PROGRAM Axis06_Status
VAR
//System_Bit
	Always_ON	:	BOOL	:=TRUE	;//상시 ON 
	Always_OFF	:	BOOL	:=FALSE	;//상시 OFF
	
	Real_Position_Data : ARRAY[0..39999] OF LREAL; // 40,000개 데이터 저장 (2초 보장)
    nIndex          : DINT := 0;                // 배열 인덱스 (0 ~ 39999)

	Axis06_Position_Read: MC_ReadActualPosition;
	Axis06_Velocity_Read: MC_ReadActualVelocity;
	nCounter: INT;
	i: INT;
	Test04: BOOL;
	Test05: BOOL;
	TEST005: BOOL;
	Axis06_Reset_01: MC_Reset;
END_VAR

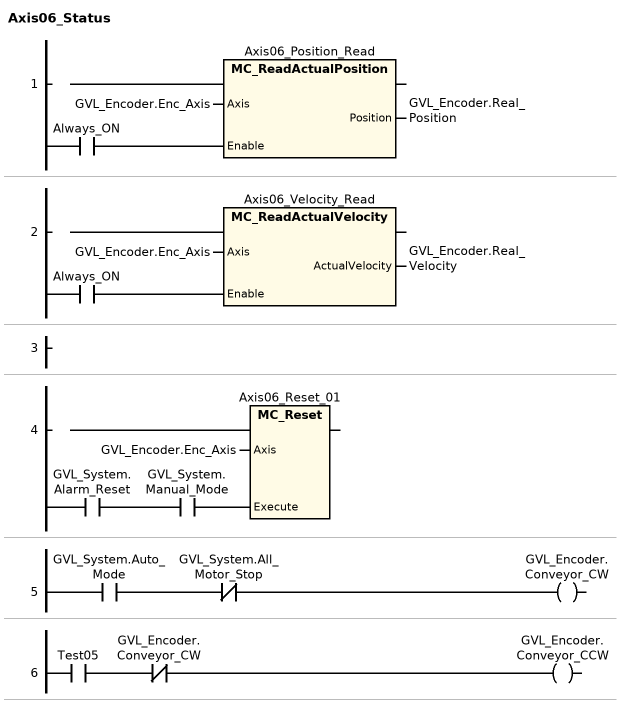
// NETWORK 1
Axis06_Position_Read(
    Axis := GVL_Encoder.Enc_Axis,
    Enable := Always_ON,
    Position => GVL_Encoder.Real_Position); // MC_ReadActualPosition

// NETWORK 2
Axis06_Velocity_Read(
    Axis := GVL_Encoder.Enc_Axis,
    Enable := Always_ON,
    ActualVelocity => GVL_Encoder.Real_Velocity); // MC_ReadActualVelocity

// NETWORK 3

// NETWORK 4
Axis06_Reset_01(Axis := GVL_Encoder.Enc_Axis, Execute := GVL_System.Alarm_Reset AND GVL_System.Manual_Mode); // MC_Reset

// NETWORK 5
GVL_Encoder.Conveyor_CW := GVL_System.Auto_Mode AND NOT GVL_System.All_Motor_Stop;

// NETWORK 6
GVL_Encoder.Conveyor_CCW := Test05 AND NOT GVL_Encoder.Conveyor_CW;

END_PROGRAM

(* stored: Version 1.1.0.1, ProductVersion 3.1.4024.15
   POU Axis06_Status: Id {08c806e5-98ff-491b-a7f7-be515b7530d8}, SpecialFunc None *)
